FUNCTION FC_SQL_InsertCommands_Encoder : STRING(255)
VAR_INPUT
    iSensorValue: INT;
    iSampleNr: INT;
END_VAR

FC_SQL_InsertCommands_Encoder := 'INSERT INTO [db_accessadmin].[Encoder] (SensorValue, SampleNr, Time) VALUES (';
FC_SQL_InsertCommands_Encoder := CONCAT(FC_SQL_InsertCommands_Encoder, INT_TO_STRING(iSensorValue));
FC_SQL_InsertCommands_Encoder := CONCAT(FC_SQL_InsertCommands_Encoder, ', ');
FC_SQL_InsertCommands_Encoder := CONCAT(FC_SQL_InsertCommands_Encoder, INT_TO_STRING(iSampleNr));
FC_SQL_InsertCommands_Encoder := CONCAT(FC_SQL_InsertCommands_Encoder, ', GETDATE());');

END_FUNCTION

(* stored: Version 1.1.0.1
   POU FC_SQL_InsertCommands_Encoder: Id {8710b876-2123-41e8-b7ca-72e97d1e6a08}, SpecialFunc None *)
